FUNCTION_BLOCK FB_ModeHandler EXTENDS FB_StateMachine IMPLEMENTS I_StateMachine
VAR_INPUT

	
	
END_VAR
VAR
	
	bStartSelftest : BOOL;
//	bStartErgonomics : BOOL;
	
	fbRightArm  : FB_ControllerArm;
	fbLeftArm  : FB_ControllerArm;
	
	eInnerState : E_ModeHandlerStates;
	
	// TODO: Move to Front end handler struct
	bRightArmEnabled_FE : BOOL;
	bLeftArmEnabled_FE : BOOL;
	bGoToIdle_FE : BOOL;
	stRightErgoCommands_FE : ST_ErgoCommands;
	stLeftErgoCommands_FE : ST_ErgoCommands;
	//----
END_VAR

OuterLopSM();

METHOD PRIVATE CheckForFailedArms : BOOL
IF fbRightArm.Failed THEN
	fbEventHandler(eNapID:=E_Event.TASK_FAILED,sTrace:=fbRightArm.EventTrace);
	fbRightArm.ErrorAck:=TRUE;
	bError := TRUE;
END_IF
IF fbLeftArm.Failed THEN
	fbEventHandler(eNapID:=E_Event.TASK_FAILED,sTrace:=fbLeftArm.EventTrace);
	fbleftArm.ErrorAck:=TRUE;
	bError := TRUE;
END_IF
END_METHOD

METHOD Disable : BOOL
VAR
	 bChildBusy : BOOL := FALSE;
END_VAR
fbRightArm(bActive:=FALSE);
fbLeftArm(bActive:=FALSE);

IF NOT fbRightArm.Ready THEN
	bChildBusy := TRUE; 
ELSIF  fbRightArm.Failed THEN
	bChildBusy := TRUE; 
	//	Stack trace and bError switching are reserved for inner loop
	fbRightArm.ErrorAck:=TRUE; // allow the arm to go Operational>DisablingInactive>Inactive
END_IF


IF NOT fbLeftArm.Ready THEN
	bChildBusy := TRUE; 
ELSIF  fbLeftArm.Failed THEN
	bChildBusy := TRUE; 
	//	Stack trace and bError switching are reserved for inner loop
	fbLeftArm.ErrorAck:=TRUE; // allow the arm to go Operational>DisablingInactive>Inactive
END_IF




IF bChildBusy THEN
	Disable := FALSE;
ELSE
	Disable := TRUE;
END_IF
END_METHOD

METHOD EnableArms : BOOL
VAR_INPUT
	
END_VAR
fbRightArm.Active:=bRightArmEnabled_FE;
fbLeftArm.Active:=bLeftArmEnabled_FE;
IF fbRightArm.Ready AND fbLeftArm.Ready THEN
	EnableArms := TRUE;
ELSE
	EnableArms := FALSE;
END_IF
END_METHOD

METHOD InnerLoopSM : BOOL
VAR
	bGoToUndocked: BOOL := FALSE;
END_VAR
// update all children FBs
ReadStatus();
fbRightArm();
fbLeftArm();

CASE CyclicInnerCase(TO_STRING(eInnerState)) OF
	E_ModeHandlerStates.Idle:
		IF bStartSelftest THEN
			IF EnableArms() THEN
				ChangeInnerState(E_ModeHandlerStates.Selftest1);
				bStartSelftest := FALSE;
			END_IF
		END_IF
		
	E_ModeHandlerStates.Selftest1:
		IF fbRightArm.Ready AND  fbLeftArm.Ready THEN
			fbRightArm.StartSelftest:=TRUE;
			fbLeftArm.StartSelftest:=TRUE;
			ChangeInnerState(E_ModeHandlerStates.Selftest2);
		ELSE
			sErrorDetails := CONCAT4('fbRightArm.bReady/fbLeftArm.bReady = ',BOOL_TO_STRING(fbRightArm.Ready),'/',BOOL_TO_STRING(fbLeftArm.Ready));
			fbEventHandler(eNapID:=E_Event.UNABLE_TO_START_TASK,sMessage:=sErrorDetails);
			bError := TRUE;
 		END_IF

	E_ModeHandlerStates.Selftest2:
		IF fbRightArm.Ready AND fbLeftArm.Ready THEN
			IF fbRightArm.Calibrated AND fbLeftArm.Calibrated THEN
				ChangeInnerState(E_ModeHandlerStates.Ergonomics1);
			ELSE
				sErrorDetails := CONCAT4('fbRightArm.Calibrated/fbLeftArm.Calibrated = ',BOOL_TO_STRING(fbRightArm.Calibrated),'/', BOOL_TO_STRING(fbLeftArm.Calibrated));				
				fbEventHandler(eNapID:=E_Event.TASK_FAILED,sMessage:=sErrorDetails);
				bError := TRUE;
			END_IF
		ELSE
			// Check/report errors from both arms
			IF fbRightArm.Failed THEN
				IF NOT fbRightArm.Docked THEN
					fbEventHandler(eNapID:=E_Event.TASK_INTERRUPTED,sTrace:=fbRightArm.EventTrace);
					fbRightArm.ErrorAck:=TRUE;
					fbRightArm.Active:=TRUE;
					bGoToUndocked := TRUE;
				ELSE
					fbEventHandler(eNapID:=E_Event.TASK_FAILED,sTrace:=fbRightArm.EventTrace);
					fbRightArm.ErrorAck:=TRUE;
					bError := TRUE;
				END_IF
			END_IF
			IF fbLeftArm.Failed THEN
				IF NOT fbLeftArm.Docked THEN
					fbEventHandler(eNapID:=E_Event.TASK_INTERRUPTED,sTrace:=fbLeftArm.EventTrace);
					fbLeftArm.ErrorAck:=TRUE;
					fbLeftArm.Active:=TRUE;
					bGoToUndocked := TRUE;
				ELSE
					fbEventHandler(eNapID:=E_Event.TASK_FAILED,sTrace:=fbLeftArm.EventTrace);
					fbleftArm.ErrorAck:=TRUE;
					bError := TRUE;
				END_IF
			END_IF
		END_IF
		IF bGoToUndocked THEN
			ChangeInnerState(E_ModeHandlerStates.SelftestUndocked);
		END_IF	
		
	E_ModeHandlerStates.SelftestUndocked:
		IF fbRightArm.Docked AND fbLeftArm.Docked THEN
			bGoToUndocked := FALSE;
			ChangeInnerState(E_ModeHandlerStates.Selftest1);
		ELSE
			// Wait... one or both arms still undocked 	
		END_IF
		
	E_ModeHandlerStates.Ergonomics1:
		IF fbRightArm.Ready AND  fbLeftArm.Ready THEN
			IF fbRightArm.Calibrated AND fbLeftArm.Calibrated THEN
				fbRightArm.StartErgonomics:=TRUE;
				fbLeftArm.StartErgonomics:=TRUE;
				ChangeInnerState(E_ModeHandlerStates.Ergonomics2);
			ELSE
				sErrorDetails := CONCAT4('fbRightArm.Calibrated/fbLeftArm.Calibrated = ',BOOL_TO_STRING(fbRightArm.Calibrated),'/', BOOL_TO_STRING(fbLeftArm.Calibrated));
				fbEventHandler(eNapID:=E_Event.UNABLE_TO_START_TASK,sMessage:=sErrorDetails);
				bError := TRUE;
			END_IF
		ELSE
			sErrorDetails := CONCAT4('fbRightArm.bReady/fbLeftArm.bReady = ',BOOL_TO_STRING(fbRightArm.Ready),'/',BOOL_TO_STRING(fbLeftArm.Ready));
			fbEventHandler(eNapID:=E_Event.UNABLE_TO_START_TASK,sMessage:=sErrorDetails);
			bError := TRUE;
 		END_IF
		
	E_ModeHandlerStates.Ergonomics2:
		bBusy := TRUE;
		IF bGoToIdle_FE THEN
			fbRightArm.StopMotors := TRUE;
			fbLeftArm.StopMotors := TRUE;
			ChangeInnerState(E_ModeHandlerStates.HaltErgonomics);
		ELSE
			IF fbRightArm.Ready AND  fbLeftArm.Ready THEN
				// Ergonomics FB is complete or failed
				// No checks for validating completeness as was in Selftest
				ChangeInnerState(E_ModeHandlerStates.Teleoperation1);
			ELSE
				fbRightArm.ErgoCommands := stRightErgoCommands_FE;
				fbLeftArm.ErgoCommands := stLeftErgoCommands_FE;	// JogInwards, JogOutwards, MovetoX, DoneErgo
				CheckForFailedArms();
			END_IF
		END_IF		
		
	E_ModeHandlerStates.HaltErgonomics:
		IF fbRightArm.Ready AND  fbLeftArm.Ready THEN
			// Ergonomics FB is complete or failed
			// No checks for validating completeness as was in Selftest
			ChangeInnerState(E_ModeHandlerStates.Idle); //Ergonomics complete, return to Idle
		ELSE 
			CheckForFailedArms();
		END_IF
		
	E_ModeHandlerStates.Teleoperation1:
		IF fbRightArm.Ready AND  fbLeftArm.Ready THEN
			IF fbRightArm.Calibrated AND fbLeftArm.Calibrated THEN
				fbRightArm.StartTeleoperation:=TRUE;
				fbLeftArm.StartTeleoperation:=TRUE;
				ChangeInnerState(E_ModeHandlerStates.Teleoperation2);
			ELSE
				sErrorDetails := CONCAT4('fbRightArm.Calibrated/fbLeftArm.Calibrated = ',BOOL_TO_STRING(fbRightArm.Calibrated),'/', BOOL_TO_STRING(fbLeftArm.Calibrated));
				fbEventHandler(eNapID:=E_Event.UNABLE_TO_START_TASK,sMessage:=sErrorDetails);
				bError := TRUE;
			END_IF
		ELSE
			sErrorDetails := CONCAT4('fbRightArm.bReady/fbLeftArm.bReady = ',BOOL_TO_STRING(fbRightArm.Ready),'/',BOOL_TO_STRING(fbLeftArm.Ready));
			fbEventHandler(eNapID:=E_Event.UNABLE_TO_START_TASK,sMessage:=sErrorDetails);
			bError := TRUE;
 		END_IF	
	
	E_ModeHandlerStates.Teleoperation2:	
		// TODO
		
	E_ModeHandlerStates.EndCase:
		ChangeInnerState(E_ModeHandlerStates.Idle);
	
END_CASE
END_METHOD

PROPERTY InnerState : UINT
GET
InnerState := THIS^.nInnerLoopState;
END_GET
END_PROPERTY

METHOD PRIVATE ReadStatus : BOOL
fbRightArm.ReadStatus();
fbLeftArm.ReadStatus();
END_METHOD

METHOD Reset : BOOL
// reset variables inherited from FB_StateMachine

(* should any of the following be reset??
bActive := FALSE;
bErrorAck := FALSE;
bAbort := FALSE;
bUserEnabled := FALSE;
*) 

// reset variables specific to this FB 
bStartSelftest := FALSE;
//bStartErgonomics := FALSE;
END_METHOD

METHOD Setup : BOOL
eStateMachineSourceID := eStateSourceID;
fbRightArm(eStateSourceID := E_StateSourceID.R_Arm,
					aErrorLog:=THIS^.aErrorLog,
					nErrorLogIndex:=THIS^.nErrorLogIndex,
					bActive := FALSE);
						
fbLeftArm(eStateSourceID := E_StateSourceID.L_Arm,
					aErrorLog:=THIS^.aErrorLog,
					nErrorLogIndex:=THIS^.nErrorLogIndex,
					bActive := FALSE);
					
SetInnerEnumeration(nStateEnum:=THIS^.eInnerState);
END_METHOD

END_FUNCTION_BLOCK

(* stored: Version 1.1.0.1, ProductVersion 3.1.4024.12
   POU FB_ModeHandler: Id {6c0947c2-5e26-462c-8382-998d509efbf9}, SpecialFunc None
   Folder HelperMethods: Id {2d12926e-8a50-48b6-9e1a-efa916a93661}
   Method CheckForFailedArms: Id {7f09cf03-80cb-4646-b0f7-89d0a85c7acc}
   Method Disable: Id {f0c33d5d-a727-4e9b-899e-99c055939f7f}
   Method EnableArms: Id {9bfb5c38-ae9a-458f-a1e8-9656e5b84026}
   Method InnerLoopSM: Id {c624c509-7772-4048-ab11-e15ae6fe4d6b}
   Property InnerState: Id {35fef907-6842-4c83-856f-001348a1b297}
   Get Get: Id {33ce7ba3-71e0-47a0-97c1-b65ea3f59f31}
   Method ReadStatus: Id {64100a46-36d6-40c5-b88c-1b41c84cb5d5}
   Method Reset: Id {94e89460-f249-45e8-8a14-69c26ac89d67}
   Method Setup: Id {22fbb005-253f-497d-af95-41c508980381} *)
